(*

.. <legal notes>

legal notes
=================
| SPDX-FileCopyrightText: © 2026 Oleksandr Tiutyk <trofimich@gmail.com>
| SPDX-License-Identifier: LGPL-3.0-only
| For details check: LGPL-3.0-only_

.. _LGPL-3.0-only: https://www.gnu.org/licenses/lgpl-3.0.en.html

.. </legal notes>

*)

FUNCTION_BLOCK ABSTRACT InputOutputDevice EXTENDS LeafAutomationComponent IMPLEMENTS IInputDevice, IOutputDevice

METHOD PROTECTED ABSTRACT OnProcessInput
END_METHOD

METHOD PROTECTED ABSTRACT OnProcessOutput
END_METHOD

METHOD FINAL ProcessInput
VAR
	exceptionCode : __SYSTEM.ExceptionCode;
	exception : TOF_Core.IException;
	exceptionReaction : TOF_Core.EXCEPTION_REACTION;
END_VAR
__TRY
	OnProcessInput();
__CATCH(exceptionCode)		
	exception := TOF_Core.ExceptionManager.GetLastException(exceptionCode);
					
	exceptionReaction := OnHandleException(exception, 'OnProcessInput');

	ProcessException(exception, exceptionReaction, "OnProcessInput error");
__ENDTRY
END_METHOD

METHOD FINAL ProcessOutput
VAR
	exceptionCode : __SYSTEM.ExceptionCode;
	exception : TOF_Core.IException;
	exceptionReaction : TOF_Core.EXCEPTION_REACTION;
END_VAR
__TRY
	OnProcessOutput();
__CATCH(exceptionCode)		
	exception := TOF_Core.ExceptionManager.GetLastException(exceptionCode);
					
	exceptionReaction := OnHandleException(exception, 'OnProcessOutput');

	ProcessException(exception, exceptionReaction, "OnProcessOutput error");
__ENDTRY
END_METHOD

END_FUNCTION_BLOCK

(* stored: Version 1.1.0.1
   POU InputOutputDevice: Id {d3cfaf06-a014-47b7-8cf6-98a0cc083f94}, SpecialFunc None
   Folder Methods to override: Id {c65c0bbf-e1ef-43ca-a18f-3c425c65c3bc}
   Method OnProcessInput: Id {94e71efd-bb71-4095-9cb0-5f4f8a38c0d8}
   Method OnProcessOutput: Id {6751103a-6dfb-417d-8b22-87cbdffa3af8}
   Method ProcessInput: Id {c8339c8d-4067-4f4a-a590-969bcf06fcfd}
   Method ProcessOutput: Id {a26c06ee-82b7-4764-95fa-cf1bbe29daa3} *)
